{attribute 'qualified_only'}
{attribute 'strict'}
TYPE DigitalOutputStatus:
(
        OFF := 0,
        ON := 1
);
END_TYPE

(* stored: Version 1.1.0.1, ProductVersion 3.1.4024.12
   DUT DigitalOutputStatus: Id {bf8724bb-82a8-44ad-9915-4228400520cc} *)
